TYPE ST_DH :
STRUCT
	dh1:ARRAY[1..4] OF REAL;
	dh2:ARRAY[1..4] OF REAL;
	dh3:ARRAY[1..4] OF REAL;
	dh4:ARRAY[1..4] OF REAL;
	dh5:ARRAY[1..4] OF REAL;
END_STRUCT
END_TYPE

(* stored: Version 1.1.0.1, ProductVersion 3.1.4024.11
   DUT ST_DH: Id {ee7523f2-f75a-4f7a-9d6a-87ebef79f4e6} *)
